# B&R Automation Studio project lab111
Automation Studio 4.5.2.102

## Configuration Config1

### Hardware
```
4PP065_0571_P74 : 4PP065.0571-P74 v1.1.2.0
  Connector IF5:
    ActivateDevice = 1
  ConfigurationID = lab111_Config1
```

## Logical view

### Library Logical/Libraries/Library (ANSIC)

#### Library.fun - Exported functions and function blocks
```iecst
{REDUND_ERROR} FUNCTION_BLOCK FB_integrator (*TODO: Add your comment here*) (*$GROUP=User,$CAT=User,$GROUPICON=User.png,$CATICON=User.png*)
	VAR_INPUT
		in : REAL;
	END_VAR
	VAR_OUTPUT
		out : REAL;
	END_VAR
	VAR
		dt : REAL;
		state : REAL;
	END_VAR
END_FUNCTION_BLOCK

{REDUND_ERROR} FUNCTION_BLOCK FB_motor (*TODO: Add your comment here*) (*$GROUP=User,$CAT=User,$GROUPICON=User.png,$CATICON=User.png*)
	VAR_INPUT
		u : REAL;
	END_VAR
	VAR_OUTPUT
		out_w : REAL;
		out_phi : REAL;
	END_VAR
	VAR
		Ke : REAL;
		Tm : REAL;
		integrator : FB_integrator;
		dt : REAL;
	END_VAR
END_FUNCTION_BLOCK

{REDUND_ERROR} FUNCTION_BLOCK FB_regulator (*TODO: Add your comment here*) (*$GROUP=User,$CAT=User,$GROUPICON=User.png,$CATICON=User.png*)
	VAR_INPUT
		e : REAL;
	END_VAR
	VAR_OUTPUT
		u : REAL;
	END_VAR
	VAR
		k_p : REAL;
		k_i : REAL;
		integrator : FB_integrator;
		iyOld : REAL;
		max_abs_value : REAL;
		dt : REAL;
	END_VAR
END_FUNCTION_BLOCK

{REDUND_ERROR} FUNCTION_BLOCK FB_integrator2 (*TODO: Add your comment here*) (*$GROUP=User,$CAT=User,$GROUPICON=User.png,$CATICON=User.png*)
	VAR_INPUT
		in : REAL;
	END_VAR
	VAR_OUTPUT
		out : REAL;
	END_VAR
	VAR
		dt : REAL;
		state : REAL;
	END_VAR
END_FUNCTION_BLOCK
```

#### FB_motor.c
```c
#include <bur/plctypes.h>
#ifdef __cplusplus
	extern "C"
	{
#endif
	#include "Library.h"
#ifdef __cplusplus
	};
#endif
/* TODO: Add your comment here */
void FB_motor(struct FB_motor* inst)
{
	REAL a = inst->u / inst->Ke - inst->out_w;
	REAL b = a / inst->Tm;

	inst->integrator.in = b;
	FB_integrator(&inst->integrator);

	inst->out_w = inst->integrator.out;
}
```

#### FB_regulator.c
```c
#include <bur/plctypes.h>
#ifdef __cplusplus
	extern "C"
	{
#endif
	#include "Library.h"
#ifdef __cplusplus
	};
#endif
/* TODO: Add your comment here */
void FB_regulator(struct FB_regulator* inst)
{
	REAL a = inst->e * inst->k_p;
	REAL b = inst->e * inst->k_i;
	a = a > inst->max_abs_value ? inst->max_abs_value : a;
	a = a < -inst->max_abs_value ? -inst->max_abs_value : a;
	inst->integrator.in = b + inst->iyOld;
	FB_integrator(&inst->integrator);
	REAL sum = a + inst->integrator.out;
	inst->u = sum;
	inst->u = inst->u >inst->max_abs_value ? inst->max_abs_value : inst->u;
	inst->u = inst->u < -inst->max_abs_value ? -inst->max_abs_value : inst->u;
	inst->iyOld = inst->u - sum;
}
```

#### FB_integrator.c
```c
#include <bur/plctypes.h>
#ifdef __cplusplus
	extern "C"
	{
#endif
	#include "Library.h"
#ifdef __cplusplus
	};
#endif
/* TODO: Add your comment here */
void FB_integrator(struct FB_integrator* inst)
{
	inst->out = inst->dt * inst->in + inst->state;
	inst->state = inst->out;
}
```

#### FB_integrator2.c
```c
#include <bur/plctypes.h>
#ifdef __cplusplus
	extern "C"
	{
#endif
	#include "Library.h"
#ifdef __cplusplus
	};
#endif
/* TODO: Add your comment here */
void FB_integrator2(struct FB_integrator2* inst)
{
	/*TODO: Add your code here*/
}
```

### Program Logical/Program

#### Variables.var
```iecst
VAR
	fb_regulator : FB_regulator;
	fb_motor : FB_motor;
	enable : BOOL;
	speed : REAL;
	counter : REAL;
	fb_motor2 : FB_motor;
END_VAR
```

#### Cyclic.c
```c
#include <bur/plctypes.h>

#ifdef _DEFAULT_INCLUDES
	#include <AsDefault.h>
#endif

void _CYCLIC ProgramCyclic(void)
{
	if (enable)
	{
		if (counter == 200)
		{
			speed = 0;
			counter++;
		}
		else if (counter == 50)
		{
			speed = 50;
		}
		if (counter < 201)
			counter++;

		fb_regulator.e = speed - fb_motor.out_w;
		FB_regulator(&fb_regulator);
		fb_motor.u = fb_regulator.u;
		fb_motor2.u = speed * fb_motor2.Ke;
		FB_motor(&fb_motor);
		FB_motor(&fb_motor2);
	}
}
```

#### Init.c
```c
#include <bur/plctypes.h>

#ifdef _DEFAULT_INCLUDES
	#include <AsDefault.h>
#endif

void _INIT ProgramInit(void)
{
	fb_motor.dt = 0.01;
	fb_motor.Ke = 0.24;
	fb_motor.Tm = 0.1;
	fb_motor.u = 0;
	fb_motor.integrator.dt = 0.01;

	fb_motor2.dt = 0.01;
	fb_motor2.Ke = 0.24;
	fb_motor2.Tm = 0.1;
	fb_motor2.u = 0;
	fb_motor2.integrator.dt = 0.01;

	fb_regulator.dt = 0.01;
	fb_regulator.integrator.dt = 0.01;
	fb_regulator.k_i = 7.2;
	fb_regulator.k_p = 0.24 * 3;
	fb_regulator.max_abs_value = 24.0;

	enable = 1;
	speed = 0;
	counter = 0;
}
```

Listed in the project but not available here: Logical/Libraries/Library/Types.typ, Logical/Libraries/Library/Constants.var
